PROGRAM _14_Config_Consum


(*s 500 sensor ampers para consumo*)
Mc._14_CONSUM.s500_Amperimetre.rAna_min:=0;
Mc._14_CONSUM.s500_Amperimetre.rAna_max:=37000;
Mc._14_CONSUM.s500_Amperimetre.rUf_min:=0;
Mc._14_CONSUM.s500_Amperimetre.rUf_max:=WORD_TO_REAL(PF_consum[2]);


Mc._14_CONSUM.rAmp:=Mc._14_CONSUM.s500_Amperimetre.rValue;

END_PROGRAM

(* stored: Version 1.1.0.1, ProductVersion 3.1.4024.10
   POU _14_Config_Consum: Id {023a7a77-0e5b-4226-b9f3-aeeae7650a83}, SpecialFunc None *)
